% RSLogix 500 project DIGITAL HEATER CONTROL.RSS, saved by version 8.30.00.16 %
PROJECT ""    % processor: Bul.1763 MicroLogix 1100 Series B %

PROGRAM FILES
  LAD 2 "MAIN"  5 rungs

DATA FILES
  O0 OUTPUT  4 elements
  I1 INPUT  6 elements
  S2 STATUS  66 elements
  B3 BINARY  1 elements
  T4 TIMER  1 elements
  C5 COUNTER  1 elements
  R6 CONTROL  1 elements
  N7 INTEGER  1 elements
  F8 FLOAT  1 elements

LADDER 2 "MAIN"
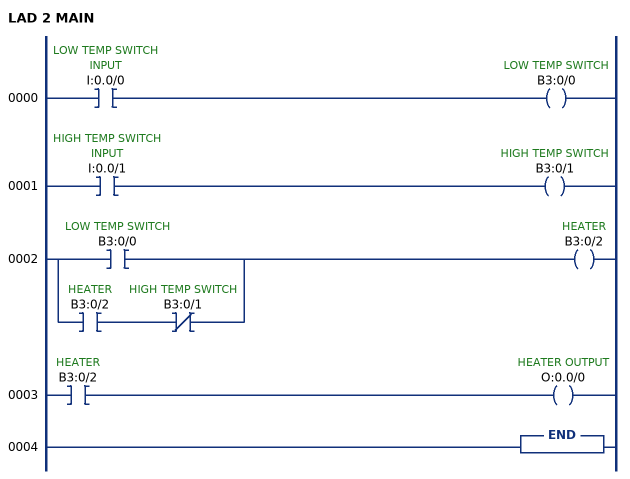
% Rung: 0 %
SOR XIC I:0.0/0 OTE B3:0/0 EOR
%   I:0.0/0  "LOW TEMP SWITCH INPUT" %
%   B3:0/0  "LOW TEMP SWITCH" %
% Rung: 1 %
SOR XIC I:0.0/1 OTE B3:0/1 EOR
%   I:0.0/1  "HIGH TEMP SWITCH INPUT" %
%   B3:0/1  "HIGH TEMP SWITCH" %
% Rung: 2 %
SOR BST XIC B3:0/0 NXB XIC B3:0/2 XIO B3:0/1 BND OTE B3:0/2 EOR
%   B3:0/0  "LOW TEMP SWITCH" %
%   B3:0/2  "HEATER" %
%   B3:0/1  "HIGH TEMP SWITCH" %
% Rung: 3 %
SOR XIC B3:0/2 OTE O:0.0/0 EOR
%   B3:0/2  "HEATER" %
%   O:0.0/0  "HEATER OUTPUT" %
% Rung: 4 %
SOR END EOR
